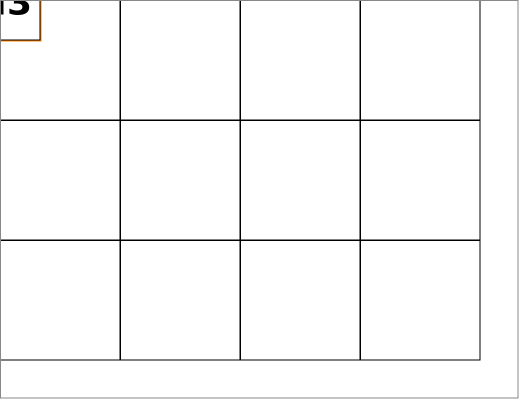
VISUALIZATION VI_Control_Xplanar  // 519x399
    Rectangle (0,0 120x120)
    Rectangle (120,0 120x120)
    Rectangle (240,0 120x120)
    Rectangle (360,0 120x120)
    Rectangle (0,120 120x120)
    Rectangle (120,120 120x120)
    Rectangle (240,120 120x120)
    Rectangle (360,120 120x120)
    Rectangle (0,240 120x120)
    Rectangle (120,240 120x120)
    Rectangle (240,240 120x120)
    Rectangle (360,240 120x120)
    Rectangle (-39,-39 80x80), "1", invisible if: NOT g_VisStationData[1].bInit
        p3560616238: g_VisStationData[1].fPosition_X/2
        p2738717112: (720-g_VisStationData[1].fPosition_Y)/2
    Rectangle (-39,-39 80x80), "2", invisible if: NOT g_VisStationData[2].bInit
        p3560616238: g_VisStationData[2].fPosition_X/2
        p2738717112: (720-g_VisStationData[2].fPosition_Y)/2
    Rectangle (-39,-39 80x80), "3", invisible if: NOT g_VisStationData[3].bInit
        p3560616238: g_VisStationData[3].fPosition_X/2
        p2738717112: (720-g_VisStationData[3].fPosition_Y)/2
    Rectangle (-39,-39 80x80), "4", invisible if: NOT g_VisStationData[4].bInit
        p3560616238: g_VisStationData[4].fPosition_X/2
        p2738717112: (720-g_VisStationData[4].fPosition_Y)/2
    Rectangle (-39,-39 80x80), "5", invisible if: NOT g_VisStationData[5].bInit
        p3560616238: g_VisStationData[5].fPosition_X/2
        p2738717112: (720-g_VisStationData[5].fPosition_Y)/2
    Rectangle (-37,-37 77x77), "M1"
        p3560616238: MAIN.fbXMotionUnit.fbMover[1].VisuPos.x/2
        p2738717112: (720-MAIN.fbXMotionUnit.fbMover[1].VisuPos.y)/2
        p2858320360: -MAIN.fbXMotionUnit.fbMover[1].VisuPos.c
    Rectangle (-37,-37 77x77), "M2"
        p3560616238: MAIN.fbXMotionUnit.fbMover[2].VisuPos.x/2
        p2738717112: (720-MAIN.fbXMotionUnit.fbMover[2].VisuPos.y)/2
        p2858320360: -MAIN.fbXMotionUnit.fbMover[2].VisuPos.c
    Rectangle (-37,-37 77x77), "M4"
        p3560616238: MAIN.fbXMotionUnit.fbMover[4].VisuPos.x/2
        p2738717112: (720-MAIN.fbXMotionUnit.fbMover[4].VisuPos.y)/2
        p2858320360: -MAIN.fbXMotionUnit.fbMover[4].VisuPos.c
    Rectangle (-37,-37 77x77), "M3"
        p3560616238: MAIN.fbXMotionUnit.fbMover[3].VisuPos.x/2
        p2738717112: (720-MAIN.fbXMotionUnit.fbMover[3].VisuPos.y)/2
        p2858320360: -MAIN.fbXMotionUnit.fbMover[3].VisuPos.c
END_VISUALIZATION

(* stored: Version 1.1.0.1
   Visu VI_Control_Xplanar: Id {d43f0dbf-72d8-4254-8a8b-664e09fa767d} *)
